TYPE ST_BoolParam :
STRUCT
  bValue      : BOOL;
  bValid      : BOOL;
  bWriteToNc  : BOOL;
END_STRUCT
END_TYPE

(* stored: Version 1.1.0.1, ProductVersion 3.1.4023.8
   DUT ST_BoolParam: Id {0c5068ec-4437-4f17-b129-c963ec451c7c} *)
